{attribute 'qualified_only'}
{attribute 'strict'}
TYPE E_Xelectrix_OperatingState :
(
	eNoDataReceived := 0,
	eOff := 1,
	eDischarge := 2,
	eCharge := 3,
	eIdle := 4
);
END_TYPE

(* stored: Version 1.1.0.1, ProductVersion 3.1.4024.6
   DUT E_Xelectrix_OperatingState: Id {9f220e87-905a-4951-9e8c-183c9652bcf6} *)
